Staubli VAL3: onRun.pgx

public program onRun(string& x_sItem[])
  local string l_sEmpty
  local num l_nResult
begin
  // execute check if need to reload
  call loadCycle(x_sItem,l_nResult)
  // execute
  call makeTraj(x_sItem)
end
